FUNCTION fLinInterpol : real
VAR_INPUT
	InputValue,Xmin,Xmax,Ymin,Ymax:REAL;
END_VAR
VAR
	b,a:REAL;
END_VAR

//y=a+bx
b:= YMin+InputValue*((Xmax-Xmin)/(Ymax-Ymin));
a:= Ymin-b*xmin;
fLinInterpol:=a+b*InputValue;

END_FUNCTION

(* stored: Version 1.1.0.1, ProductVersion 3.1.4024.6
   POU fLinInterpol: Id {5ea7fabf-9bde-409d-a780-f61b770ee3e9}, SpecialFunc None *)
